(*
Nazwa:			FB_CatchStation
Opis:			Chwytak pod stacjami 
Wersja:			v1.2
Data:			2025-07-08
Autor:			TW,DP
Urzadzenia:		Silownik chwytania, podnośnik JIESANG
Konfiguracja:	
Zmiany:
20250708 - Homing false po wyj. z Manual
20230222 - Zwieksozmny czas bledu 9

Info:
- dodano błędy od nastaw powyżej max i min (error 7 i 8)
- dodawno bHomingNeeded
- wylaczanie wyjść zmiana 2 wylaczanie wyjsc jak zniknie Enable
*)


FUNCTION_BLOCK FB_CatchStation
VAR_INPUT
	bEnable: BOOL;						//Zezwolenie na pracę
	bEStop:BOOL;						//Stop Awaryjny włączony
	bRun:BOOL;							//Rozkaz łapania 
	bHoming:BOOL;						//Zezwolenie na wykonanie bazowania i pozycjonowania podajnika
	bHeightSet:BOOL;					//Ustaw wysokość
	bChangeover:BOOL;					//Ustawianie na zadaną wysokość do wymiany elementów formatowych
	bChangeOver2:BOOL;
	bIgnoreError:BOOL;					//Ignorowania błędów cyklu pracy
	bReset:BOOL;						//Reset błędu, jeśli w stanie "eError"
	nGripperScrewerPosition   	:LREAL; // Aktualna pozycja serwa od podnoszenia
	nSafetyScrewerPosition		:LREAL;	// zadana bezpieczna pozycja 
	bScrewerbError				:BOOL;  // Sygnał błędu od zakręcarki
	nPositionHeightSV:LREAL;			//Wysokość zadana na której ma znajdować się stacja
	bOpenedActuatorSensor:BOOL;			//Czujnik otwarcia siłownika łapania
	bClosedActuatorSensor:BOOL;			//Czujnik otwarcia siłownika łapania
	lrMaxHeight:LREAL;					//Maksymalna wysokość podnośnika chwytaka
	lrMinHeight:LREAL;					//Minimalna wysokość podnośnika chwytaka
	bManualMovement:BOOL;				//Zezwolenie na ruchy ręcznę
	bUnlockColision:BOOL:=FALSE;		//Odblokowywanie możliwośći kolizji
	bAlarmSVCVDiffHeightDisable:BOOL;	//Wyłączenie alarmu od rożnicy wysokości zadanej od aktualnej
	bNoLifter:BOOL;						//Podnośnik
	
	_HEIGHTMOTOR_ :BOOL;	
				
	rHeightMotorPositionOffset :REAL;		//Wysokość bazowani podnośnika
	udiHeightMotorEncoderCV		: UDINT;
	bHeightEncoderSetCDone		: BOOL;	

	_ALARMINFO_ :BOOL;
	iStationIndex:UDINT;					//Numer stacji 
	sStationName:WSTRING;					//Nazwa stacji	

	
END_VAR
VAR_OUTPUT
	eState: E_Station;						//Stan ogólny bloku
	eRunningState: E_CatchStationState;		//Stan wewnętrzny
	bError: BOOL;							//Błąd stacji
	nErrorNr: UDINT;						//Nr błędu podajnika platynek
	sErrorDescription:STRING(200);				//Opis błędu
	sErrorDescription2: STRING(200);				//Opis błędu 2
	sErrorStationName:STRING;				//Nazwa stacji
	udiStationID: UDINT;				// Nr stacji

	bCatchActuator:BOOL;					//Sterownie siłownika łapania opakowania
	bHeightMotorUp:BOOL;					//Sterowanie silnikiem podnośnika  - RUCH W GÓRĘ
	bHeightMotorDown:BOOL;					//Sterowanie silnikiem podnośnika  - RUCH W DÓŁ
	lrHeightMotorCV:LREAL;					//Aktualna pozycja podnośnika
	tCycleTime:TIME;
	bHomingDone:BOOL;						//Wymagane ponowne bazowanie (blad podczas bazowania lub stop awaryjny)
	bCycleDone:BOOL;
	bCycleNotDone:BOOL;
	
				
	udiHeightMotorEncoderSetCV	: UDINT;	
	bHeightEncoderSetC			: BOOL;		

END_VAR
VAR
	tonHeightNoChange: TON; 			//Timer wykrycia braku ruchu siłownika zmiany wysokości stacji
	nLastPositionHeightCV: LREAL;		//Pozycja podnośnika w poprzednim cyklu programu
	tonErrorHeightChange: TON; 			//Timer błędu podnośnika
	// Czas zadziałania siłownika
	tonCatchingTime: TON;
	// Timer blokady otwierania chwytaka
	tonOpeningBlocked: TON;
	rtEncoderHomed:R_TRIG;
	tonCycleTimer:TON;
	rtrigCycleTimerRead:R_TRIG;
	
	tofMotorUpPermition: TOF;
	tofMotorDownPermition: TOF;
	tonLimitPosMinReachedDelay: TON;
	tonLimitPosMaxReachedDelay: TON;
	tonMaxHeight		: TON;
	tonMinHeight		: TON;
	tonSVCVDiffHeight	: TON;
	
	//Podnośnik Jiesang	
	fbHeightMotorEncoder: FB_JiesangActuatorEncoderModul;	// Blok enkodera podnośnika chwytaka stabilizującego pod zakręcarką	
	bHeightMotorEncoderCounterReset:BOOL; 				//Sygnał resetu enkodera
	bHeightMotorEncoderHomed:BOOL;						//Informacja od enkodera że jest zbazowany

	eLastState: E_Station;							//Stan ogólny bloku
	eLastRunningState: E_CatchStationState;			//Stan podbloku
	eLastStateTemp: E_Station;						//Stan ogólny bloku
	eLastRunningStateTemp: E_CatchStationState;		//Stan podbloku
	bStateError: BOOL;

	tonStopping: TON;
	tofHeightMotorDown: TOF;
	iCaseChangeover: INT;
	tonChangeOverLimitPosMinReachedDelay: TON;
	tonChangeoverLimitPosMaxReachedDelay: TON;
	
	//Zmienne od EVENTLOGGER
	bAlarmInit 						: BOOL := TRUE; 
	nAlarmNumerator					: INT;
	arfbAlarm						: ARRAY[0..19] OF  FB_TcAlarm;		//Tablica bloczków błędów
	fbSourceInfo 					: FB_TcSourceInfo;
	iSourceInfo						: I_TcSourceInfo;
	sAlarmTest						: STRING;
	//Koniec zmiennych od EVENTLOGGER
END_VAR

VAR_IN_OUT
	bManualCatchActuator:BOOL;		//Ruch ręczny siłownikiem podajnika platynek
	bManualHeightMotorUp:BOOL;			//Ruch ręczny podnośnika stacji w górę
	bManualHeightMotorDown:BOOL;		//Ruch ręczny podnośnika stacji w dół
END_VAR

HeightMotor();
ErrorHandling();
Control();
Changeover();
Statistics();
aStationID();
(*Zapisywanie ostatniego stanu*)
IF eLastStateTemp<>eState THEN
	eLastState := eLastStateTemp;
END_IF
eLastStateTemp := eState;
IF eLastRunningStateTemp<>eRunningState THEN
	eLastRunningState := eLastRunningStateTemp;
END_IF
eLastRunningStateTemp := eRunningState;
(*Koniec Zapisywanie ostatniego stanu*)


nLastPositionHeightCV:=lrHeightMotorCV;

ACTION aStationID:
udiStationID	:=	iStationIndex;
END_ACTION

ACTION Changeover:
tonChangeOverLimitPosMinReachedDelay(IN:=(lrHeightMotorCV<=lrMinHeight) AND bChangeover,PT:=T#2S);
tonChangeoverLimitPosMaxReachedDelay(IN:=(lrHeightMotorCV>=lrMaxHeight) AND bChangeover,PT:=T#2S);


//Przeniesione do PreparingToDisabled
(*CASE iCaseChangeover OF
	
	0: //Włączenie ustawiania
		IF bChangeover THEN
			iCaseChangeover := iCaseChangeover + 10;
			bHeightMotorDown:=FALSE;
			bHeightMotorUp:=FALSE;
		END_IF
		
	10: //Ustawianie stacji na wysokość 
		IF bHeightMotorEncoderHomed THEN
			bHeightMotorEncoderCounterReset	:=	FALSE;
			bHeightMotorUp					:=	lrHeightMotorCV	<=	200;
			bHeightMotorDown				:=	lrHeightMotorCV	>=	200;
			//Kiedy stacja osiągnie wysokość zadaną
			IF ABS(lrHeightMotorCV-nPositionHeightSV)<2 OR tonChangeoverLimitPosMaxReachedDelay.Q OR tonChangeOverLimitPosMinReachedDelay.Q  THEN
				bHeightMotorDown			:=	FALSE;
				bHeightMotorUp				:=	FALSE;
				iCaseChangeover 			:=	iCaseChangeover + 10;
			END_IF			
		ELSE
			bHeightMotorDown		:=	FALSE;
			bHeightMotorUp			:=	FALSE;
			iCaseChangeover 		:=  0;
		END_IF	
		
	20: //Czekanie na wyłączenie przezbrajania i ustawienie na odpowiednią wysokość z receptury
			IF NOT bChangeover THEN
				iCaseChangeover := iCaseChangeover + 10;
			END_IF
	30: //Ustawianie stacji na wysokość z receptury
		IF bHeightMotorEncoderHomed THEN
			bHeightMotorEncoderCounterReset	:=	FALSE;
			bHeightMotorUp					:=	lrHeightMotorCV	<=	nPositionHeightSV;
			bHeightMotorDown				:=	lrHeightMotorCV	>=	nPositionHeightSV;
			//Kiedy stacja osiągnie wysokość zadaną
			IF ABS(lrHeightMotorCV-nPositionHeightSV)<2 OR tonChangeoverLimitPosMaxReachedDelay.Q OR tonChangeOverLimitPosMinReachedDelay.Q  THEN
				bHeightMotorDown			:=	FALSE;
				bHeightMotorUp				:=	FALSE;
				iCaseChangeover 			:=	iCaseChangeover + 10;
			END_IF			
		ELSE
			bHeightMotorDown		:=	FALSE;
			bHeightMotorUp			:=	FALSE;
			iCaseChangeover 		:=  0;
		END_IF
	40: //Ustawianie stacji na wysokość z receptury	
		iCaseChangeover 		:=  0;

END_CASE
*)
END_ACTION

ACTION Control:

	(** TIMERY**)
	rtEncoderHomed(CLK:=bHeightMotorEncoderHomed,Q=>);
	tonHeightNoChange(IN:=((bHeightMotorUp OR bHeightMotorDown) AND (nLastPositionHeightCV=lrHeightMotorCV)), PT:=T#1S); 
	tonLimitPosMinReachedDelay(IN:=(lrHeightMotorCV<=lrMinHeight) AND eState=E_Station.eHoming,PT:=T#2S);
	tonLimitPosMaxReachedDelay(IN:=(lrHeightMotorCV>=lrMaxHeight) AND eState=E_Station.eHoming,PT:=T#2S);
	tonStopping(IN:=eState=E_Station.eStopping,PT:=T#2S);
	tofMotorUpPermition(IN:=bHeightMotorDown,PT:=T#250MS);
	tofMotorDownPermition(IN:=bHeightMotorUp ,PT:=T#250MS);	
	(*****Wyłączenie enable*****)
	IF NOT bEnable OR bChangeover THEN //Lub przezbrajania
		IF eState <> E_Station.eDisabled AND eState <> E_Station.ePreparingToDisable AND nGripperScrewerPosition>nSafetyScrewerPosition AND NOT bScrewerbError THEN
				eState 				:= E_Station.ePreparingToDisable; 
		END_IF	
	END_IF

	(*****Estop*****)
	IF NOT bEstop  THEN	
		IF eState <> E_Station.eAborted AND eState <> E_Station.eAborting AND eState <> E_Station.eDisabled THEN
				eState 				:= E_Station.eAborting; 
		END_IF
	END_IF

	CASE eState OF
	/////////////////////////////	
		E_Station.eDisabled: 					// Stan nieaktywnosci (Stacja wyłączona) 

			IF bEnable THEN
				eState 				:= E_Station.ePreparingToReady; 
			END_IF 
			
    /////////////////////////////	    
		E_Station.eAborted: 					// Stan bezpiecznego zatrzymania (po Abortingu) 

			IF bEStop THEN
				eState 				:= E_Station.ePreparingToReady;
			END_IF
			
	/////////////////////////////	
		E_Station.eAborting:                 	// Stan bezpiecznego zatrzymywania (po EStopie)

			bHeightMotorUp				:=	FALSE;
			bHeightMotorDown			:=	FALSE;
			eState := E_Station.eAborted;  
			eRunningState:=E_CatchStationState.eDisabled;
			
	/////////////////////////////			
		E_Station.eError:                 	 	// Stan błędu 	

			iCaseChangeover 		:=	0;
			IF bReset THEN
				eState 				:=	E_Station.eResetting;
			END_IF
						
	/////////////////////////////
		E_Station.eResetting:					// Stan resetowania bledu (po Errorze)
	
			bError := FALSE;

			IF NOT bError THEN
				nErrorNr 			:=	0;
   				sErrorDescription 	:=	'';
				eState 				:=	E_Station.ePreparingToReady;
			ELSE
				eState 				:=	E_Station.eError;
			END_IF
        
	/////////////////////////////
		E_Station.eManualMovement:     			// Stan ruchów manualnych  

			ManualMovements();
			//Wyjście z trybu serwisowego
			IF NOT bManualMovement THEN
				IF bHomingDone AND ABS(lrHeightMotorCV - nPositionHeightSV)> 2 THEN
					bHomingDone := FALSE;
				END_IF
				bCatchActuator				:=	FALSE;
				bHeightMotorUp				:=	FALSE;
				bHeightMotorDown			:=	FALSE;
				bManualCatchActuator		:=	bCatchActuator;
				eState:=E_Station.eReady;
			END_IF

	/////////////////////////////
		E_Station.eHoming:						// Stan bazowania 
	IF (nGripperScrewerPosition>nSafetyScrewerPosition AND NOT bScrewerbError) OR bManualMovement THEN  // co to za bzdura
			Homing();
			IF NOT bHoming AND NOT bHeightSet THEN // co to za bzdura
			   eState:=E_Station.ePreparingToReady;
			   	bHeightMotorDown:=FALSE;
				bHeightMotorUp:=FALSE;
			END_IF		
	END_IF		
	/////////////////////////////
		E_Station.eHomingDone:                  // Stan wykonania bazowania 
	
			bHeightMotorDown					:=	FALSE;
			bHeightMotorUp						:=	FALSE;
			bHeightMotorEncoderCounterReset		:=	FALSE;
			bHomingDone							:=	TRUE;
			IF NOT bHoming AND NOT bHeightSet THEN
			   eState:=E_Station.eReady;
			END_IF
			
	/////////////////////////////
		E_Station.ePreparingToReady:            // Stan przygotowywania do gotowosci (zawsze przed Ready)  
	
			bCatchActuator	:=	FALSE;
			eRunningState	:=	E_CatchStationState.eReady;
			eState			:=	E_Station.eReady;	
			
	/////////////////////////////
		E_Station.ePreparingToDisable:          // Stan przygotowywania do nieaktywnosci (po wyłączeniu Enable) 
  
			bCatchActuator:=FALSE;
			IF NOT bChangeOver THEN //Normalne wyłączenie
				bHeightMotorUp:=TRUE;
				bHeightMotorDown:=FALSE;	
				IF tonHeightNoChange.Q THEN
					bHeightMotorUp:=FALSE;
					eState:=E_Station.eDisabled;
					eRunningState:=E_CatchStationState.eDisabled;
				END_IF	
			ELSE //Wyłączenie z przebrajaniem na pozycje 200
				IF bHeightMotorEncoderHomed THEN
					bHeightMotorEncoderCounterReset	:=	FALSE;
					bHeightMotorUp					:=	lrHeightMotorCV	<=	150 AND NOT tofMotorUpPermition.Q;
					bHeightMotorDown				:=	lrHeightMotorCV	>=	150 AND NOT tofMotorDownPermition.Q;
					//Kiedy stacja osiągnie wysokość zadaną
					IF ABS(lrHeightMotorCV-150)<2 OR tonChangeoverLimitPosMaxReachedDelay.Q OR tonChangeOverLimitPosMinReachedDelay.Q  THEN
						bHeightMotorDown			:=	FALSE;
						bHeightMotorUp				:=	FALSE;
						eState						:=	E_Station.eDisabled;
						eRunningState				:=	E_CatchStationState.eDisabled;
					END_IF			
				ELSE
					bHeightMotorDown				:=	FALSE;
					bHeightMotorUp					:=	FALSE;
					eState								:=E_Station.eDisabled;
					eRunningState					:=	E_CatchStationState.eDisabled;
				END_IF	
			END_IF
				
	/////////////////////////////
		E_Station.eReady:						// Stan gotowosci 

			IF bRun AND NOT bCycleDone AND NOT bCycleNotDone THEN
				eState 				:= E_Station.eStarting; 
			END_IF
			IF bHoming OR bHeightSet OR bChangeover THEN
				eState 				:= E_Station.eHoming; 
			END_IF
			IF bManualMovement THEN
				//Jeśli przejście w tryb ruchów manualnych przepisz wszystkie stany siłowników sterowanych przez moduł
				//aby zapobiec ewentualnym kolizjom po wejściu w tryb serwisowy
				bManualCatchActuator		:= bCatchActuator;
				bManualHeightMotorUp		:= bHeightMotorUp;
				bManualHeightMotorDown		:= bHeightMotorDown;
				
				eState 						:= E_Station.eManualMovement; 
				eRunningState 				:= E_CatchStationState.eReady;
 
			END_IF
			IF NOT bRun THEN
				bCycleDone 			:= FALSE;
				bCycleNotDone 		:= FALSE;			
			END_IF
			
	/////////////////////////////
		E_Station.eStopping:					// Stan zatrzymywania 
					
			Running();
			IF bOpenedActuatorSensor OR tonStopping.Q THEN //NEW
				eState						:=	E_Station.eReady;
				eRunningState 				:=	E_CatchStationState.eReady;
			END_IF
			
	/////////////////////////////
		E_Station.eStarting:                  	// Stan uruchamiania (po Ready)
				
			eState					 := E_Station.eRunning; 

	/////////////////////////////
		E_Station.eRunning:               		// Stan wykonywania cyklu (po Startingu), w tym stanie osobny

			Running();
			IF NOT bRun THEN 					(*Przerywanie cyklu*)
				eState				:= E_Station.eStopping;
				bCycleNotDone		:= TRUE;
			END_IF
			(*IF bCycleDone OR bCycleNotDone THEN (*Cykl zakończony*)
				eState 				 := E_Station.eReady;
			END_IF*)						
		ELSE
		
		
	/////////////////////////////		
	END_CASE
END_ACTION

ACTION ErrorHandling:
// Alarm_0440	440	Error	Blokada otwarcia chwytaka - sprawdź czujnik
// Alarm_0441	441	Error	Blokada podnośnika lub brak zasilania - sprawdź czujnik lub odblokuj mechanicznie
// Alarm_0442	442	Error	Wartość zadana wysokości jest większa od maksymalnej - zmień ustawienia w recepturze {0}
// Alarm_0443	443	Error	Wartość zadana wysokości jest mniejsza od minimalnej - zmień ustawienia w recepturze {0}
// Alarm_0444	444	Error	Wartość aktualna jest zbyt różna od zadanej - zmień ustawienia w recepturze lub ustaw stację

IF bAlarmInit THEN
    bAlarmInit := FALSE; 
	fbSourceInfo.Clear();
	fbSourceInfo.sName:=wsLiteral_TO_UTF8(sStationName);//'Machine';
	fbSourceInfo.nId:=iStationIndex;//2700;
	// Alarm_0440	440	Error	Blokada otwarcia chwytaka - sprawdź czujnik
    arfbAlarm[0].CreateEx(stEventEntry := TC_EVENTS.AlarmClass.Alarm_0440, bWithConfirmation:= FALSE,  ipSourceInfo:= fbSourceInfo); 
	// Alarm_0441	441	Error	Blokada podnośnika lub brak zasilania - sprawdź czujnik lub odblokuj mechanicznie
	arfbAlarm[1].CreateEx(stEventEntry := TC_EVENTS.AlarmClass.Alarm_0441, bWithConfirmation:= FALSE,  ipSourceInfo:= fbSourceInfo);
	// Alarm_0442	442	Error	Wartość zadana wysokości jest większa od maksymalnej - zmień ustawienia w recepturze {0}
	arfbAlarm[2].CreateEx(stEventEntry := TC_EVENTS.AlarmClass.Alarm_0442, bWithConfirmation:= FALSE,  ipSourceInfo:= fbSourceInfo);
	// Alarm_0443	443	Error	Wartość zadana wysokości jest mniejsza od minimalnej - zmień ustawienia w recepturze {0}
	arfbAlarm[3].CreateEx(stEventEntry := TC_EVENTS.AlarmClass.Alarm_0443, bWithConfirmation:= FALSE,  ipSourceInfo:= fbSourceInfo);
	// Alarm_0444	444	Error	Wartość aktualna jest zbyt różna od zadanej - zmień ustawienia w recepturze lub ustaw stację
	arfbAlarm[4].CreateEx(stEventEntry := TC_EVENTS.AlarmClass.Alarm_0444, bWithConfirmation:= FALSE,  ipSourceInfo:= fbSourceInfo);
END_IF

//OBSŁUGA BŁĘDÓW PODAJNIKA PLATYNEK

//************LISTA BŁĘDÓW***************
bStateError:= (eState=E_Station.eError) OR (eState=E_Station.eResetting) OR bIgnoreError;




IF bEnable THEN
	// Alarm_0440	440	Error	Blokada otwarcia chwytaka - sprawdź czujnik
	//Error 1 - Blokada otwarcia chwytaka
	tonOpeningBlocked(IN:=NOT bCatchActuator AND NOT bOpenedActuatorSensor, PT:=T#3S);
	
	IF tonOpeningBlocked.Q THEN
		IF NOT arfbAlarm[0].bActive THEN
			arfbAlarm[0].Raise(nTimeStamp:=0);
		END_IF
	ELSE	
		IF  arfbAlarm[0].bActive AND bReset THEN
			arfbAlarm[0].Clear(nTimeStamp:=0, bResetConfirmation:= FALSE);
		END_IF
// 		sErrorDescription:='Blokada otwarcia chwytaka - sprawdź czujnik';
// 		bHeightMotorUp:=FALSE;
// 		bError := TRUE;
// 		nErrorNr:=281;	
// 		//nErrorNr := nErrorNr+iStationIndex;
	END_IF
	// Alarm_0441	441	Error	Blokada podnośnika lub brak zasilania - sprawdź czujnik lub odblokuj mechanicznie
	//Error 2 - podnośnik nie porusza się pomimo wysterowania 
	tonErrorHeightChange(IN:=(bHeightMotorUp OR bHeightMotorDown) AND nLastPositionHeightCV=lrHeightMotorCV AND NOT bNoLifter, PT:=T#3S);
	
	IF tonErrorHeightChange.Q THEN
		IF NOT arfbAlarm[1].bActive THEN
			bHeightMotorUp:=FALSE;
			bHeightMotorDown:=FALSE;
			arfbAlarm[1].Raise(nTimeStamp:=0);
		END_IF
	ELSE	
		IF  arfbAlarm[1].bActive AND bReset THEN
			arfbAlarm[1].Clear(nTimeStamp:=0, bResetConfirmation:= FALSE);
		END_IF
// 		bHeightMotorUp:=FALSE;
// 		bHeightMotorDown:=FALSE;
// 		bError := TRUE;
// 		nErrorNr:=282;
// 		//nErrorNr := nErrorNr+iStationIndex;
// 		sErrorDescription:='Blokada podnośnika lub brak zasilania - sprawdź czujnik lub odblokuj mechanicznie';	
	END_IF
	
	// Alarm_0442	442	Error	Wartość zadana wysokości jest większa od maksymalnej - zmień ustawienia w recepturze {0}
	//Error 3 - Bład nastaw max
	tonMaxHeight(IN:=nPositionHeightSV>lrMaxHeight+1 AND bHomingDone AND lrMaxHeight>0 AND eState=E_Station.eReady,PT:=T#30S);
	IF tonMaxHeight.Q THEN
		arfbAlarm[2].ipArguments.Clear() .AddLReal(lrMaxHeight);
		IF NOT arfbAlarm[2].bActive THEN
			bHeightMotorUp:=FALSE;
			bHeightMotorDown:=FALSE;
			arfbAlarm[2].Raise(nTimeStamp:=0);
		END_IF
	ELSE	
		IF  arfbAlarm[2].bActive AND bReset THEN
			arfbAlarm[2].Clear(nTimeStamp:=0, bResetConfirmation:= FALSE);
		END_IF	
// 		bHeightMotorUp:=FALSE;
// 		bHeightMotorDown:=FALSE;
// 		bError := TRUE;
// 		nErrorNr:=283;
// 		//nErrorNr := nErrorNr+iStationIndex;
// 		sErrorDescription:='Wartość zadana wysokości jest większa od maksymalnej - zmień ustawienia w recepturze';
// 		sErrorDescription2:=REAL_TO_STRING(LREAL_TO_INT(lrMaxHeight));
	END_IF
	// Alarm_0443	443	Error	Wartość zadana wysokości jest mniejsza od minimalnej - zmień ustawienia w recepturze {0}
	//Error 4 - Bład nastaw min
	tonMinHeight(IN:=nPositionHeightSV<lrMinHeight-1 AND bHomingDone AND lrMinHeight>0 AND eState=E_Station.eReady,PT:=T#30S);
	IF tonMinHeight.Q THEN
		arfbAlarm[3].ipArguments.Clear() .AddLReal(lrMinHeight);
		IF NOT arfbAlarm[3].bActive THEN
			bHeightMotorUp:=FALSE;
			bHeightMotorDown:=FALSE;
			arfbAlarm[3].Raise(nTimeStamp:=0);
		END_IF
	ELSE	
		IF  arfbAlarm[3].bActive AND bReset THEN
			arfbAlarm[3].Clear(nTimeStamp:=0, bResetConfirmation:= FALSE);
		END_IF
// 		bHeightMotorUp:=FALSE;
// 		bHeightMotorDown:=FALSE;
// 		bError := TRUE;
// 		nErrorNr:=284;
// 		//nErrorNr := nErrorNr+iStationIndex;
// 		sErrorDescription:='Wartość zadana wysokości jest mniejsza od minimalnej - zmień ustawienia w recepturze ';
// 		sErrorDescription2:=REAL_TO_STRING(LREAL_TO_INT(lrMinHeight));
	END_IF
	// Alarm_0444	444	Error	Wartość aktualna jest zbyt różna od zadanej - zmień ustawienia w recepturze lub ustaw stację
	//Error 5 - Bład zbyt dużej różnicy nastaw
	//tonSVCVDiffHeight(IN:=ABS(nPositionHeightSV-lrHeightMotorCV)>10 AND bHomingDone AND NOT bAlarmSVCVDiffHeightDisable AND eState=E_Station.eReady AND NOT bChangeOver2,PT:=T#5M);
	IF tonSVCVDiffHeight.Q THEN
		arfbAlarm[4].ipArguments.Clear() .AddLReal(nPositionHeightSV);
		IF NOT arfbAlarm[4].bActive THEN
			bHeightMotorUp:=FALSE;
			bHeightMotorDown:=FALSE;
			arfbAlarm[4].Raise(nTimeStamp:=0);
		END_IF
	ELSE	
		IF  arfbAlarm[4].bActive AND bReset THEN
			arfbAlarm[4].Clear(nTimeStamp:=0, bResetConfirmation:= FALSE);
		END_IF
// 		bHeightMotorUp:=FALSE;
// 		bHeightMotorDown:=FALSE;
// 		bError := TRUE;
// 		nErrorNr:=285;
// 		//nErrorNr := nErrorNr+iStationIndex;
// 		sErrorDescription:='Wartość aktualna jest zbyt różna od zadanej - zmień ustawienia w recepturze lub ustaw stację';
// 		sErrorDescription2:=REAL_TO_STRING(LREAL_TO_INT(nPositionHeightSV));
		
	END_IF	
		
	
	
ELSE
	bError := FALSE;
END_IF

	
//******************PRZEJŚCIE DO eERROR*****************************

IF bError AND NOT bStateError THEN
	IF eLastState = eRunning THEN
		bCycleNotDone := TRUE;
	END_IF
	eState := E_Station.eError;
END_IF

//****************WYŚWIETLANIE STATUSU BLEDU***********************

(*Wyświetlanie błedu na wyjściu*)
bError							:= FALSE;
FOR nAlarmNumerator := 0 TO 19 DO
	bError						:= bError OR arfbAlarm[nAlarmNumerator].bActive;
END_FOR

(*Przepisywanie nazwy stacji*)
sErrorStationName := WSTRING_TO_STRING(sStationName);


//Jezeli nie zbazowane to potrzebne bazowanie
IF NOT bHeightMotorEncoderHomed AND NOT bNoLifter  THEN
	bHomingDone:=FALSE;
END_IF
END_ACTION

ACTION HeightMotor:
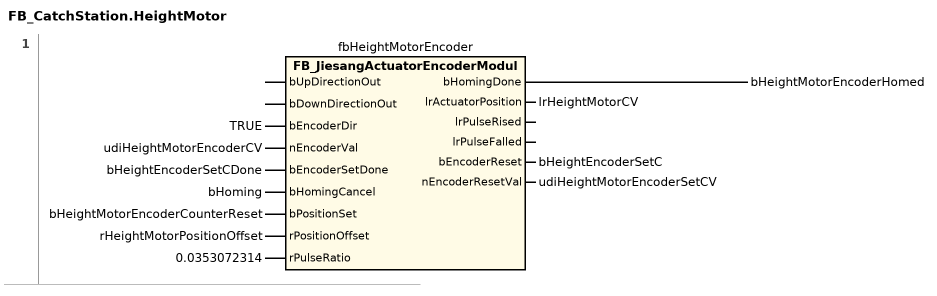
// NETWORK 1
fbHeightMotorEncoder(
    bEncoderDir := TRUE,
    nEncoderVal := udiHeightMotorEncoderCV,
    bEncoderSetDone := bHeightEncoderSetCDone,
    bHomingCancel := bHoming,
    bPositionSet := bHeightMotorEncoderCounterReset,
    rPositionOffset := rHeightMotorPositionOffset,
    rPulseRatio := 0.0353072314,
    lrActuatorPosition => lrHeightMotorCV,
    bEncoderReset => bHeightEncoderSetC,
    nEncoderResetVal => udiHeightMotorEncoderSetCV); // FB_JiesangActuatorEncoderModul
bHeightMotorEncoderHomed := fbHeightMotorEncoder.bHomingDone;
END_ACTION

ACTION Homing:
//BAZOWANIE
bCatchActuator:=FALSE;
	
//Uwaga nie zmieniać czasu bo jednocześnie dwie stację jadą do góry
tofHeightMotorDown(IN:=bHeightMotorDown, PT:=T#1S); //Zabezpieczenie przed zbyt szybkim przełączeniem pomiędzy Down a Up, bezpiecznieki sie palą, 


//Podnoszenie stacji do maksymalnej pozycji
IF NOT bHeightMotorEncoderHomed OR rtEncoderHomed.Q THEN
	bHeightMotorUp:=(*TRUE*) NOT tofHeightMotorDown.Q;;
	bHeightMotorDown:=FALSE;
	IF tonHeightNoChange.Q THEN
		bHeightMotorEncoderCounterReset:=TRUE;
		bHeightMotorUp:=FALSE;
	END_IF
	//Jesli enkoder zbazowany zakończ bazowanie	
	IF rtEncoderHomed.Q THEN
		bHeightMotorUp:=FALSE;
		bHeightMotorDown:=FALSE;
		eState:=E_Station.eHomingDone;
	END_IF		
		
//Po podniesieniu stacji opuszczanie do ustalonej wysokości
ELSIF bHeightMotorEncoderHomed THEN
	bHeightMotorEncoderCounterReset:=FALSE;
	bHeightMotorUp:=lrHeightMotorCV<=nPositionHeightSV;
	bHeightMotorDown:=lrHeightMotorCV>=nPositionHeightSV (*AND lrHeightMotorCV>=lrMinHeight*);
	//Kiedy stacja osiągnie wysokość zadaną
	IF ABS(lrHeightMotorCV-nPositionHeightSV)<1 OR tonLimitPosMaxReachedDelay.Q OR tonLimitPosMinReachedDelay.Q (*OR lrHeightMotorCV>=lrMinHeight*) THEN
		bHeightMotorDown:=FALSE;
		bHeightMotorUp:=FALSE;
		eState:=E_Station.eHomingDone;
	END_IF			
END_IF

	
//Opcja braku podnośnika	
IF bNoLifter THEN
	eState:=E_Station.eHomingDone;
END_IF
END_ACTION

ACTION ManualMovements:

//W trybie ruchów manualnych wykonuj ruchy za pomocą rozkazów manualnych
IF NOT bRun THEN
	bCatchActuator:=bManualCatchActuator;
	bHeightMotorUp:=bManualHeightMotorUp;
	bHeightMotorDown:=bManualHeightMotorDown;
ELSE	//Kasuje zeby po cyklu nic sie nie poruszało
	bManualCatchActuator := FALSE;
	bManualHeightMotorUp  := FALSE;
	bManualHeightMotorDown  := FALSE;
END_IF


IF bHoming OR bHeightSet THEN
	eState:=E_Station.eHoming;
END_IF
	
Running();
	
//Zabezpieczenie przed kolizją stacji poprzez ruch podnośnika	
IF bHeightMotorDown AND lrHeightMotorCV<=lrMinHeight AND NOT bHoming AND NOT bHeightSet THEN
	bHeightMotorDown:=FALSE;
END_IF	

IF bHeightMotorUp AND lrHeightMotorCV>=lrMaxHeight AND NOT bHoming AND NOT bHeightSet THEN
	bHeightMotorUp:=FALSE;
END_IF		 

IF NOT bRun THEN
	bCycleDone 					:= FALSE;
	bCycleNotDone 				:= FALSE;	
END_IF
END_ACTION

ACTION Running:

//Timery
tonCatchingTime(IN:=(eRunningState=E_CatchStationState.eCatching), PT:=T#500MS);


CASE eRunningState OF
	
	//NIEGOTOWY
	E_CatchStationState.eDisabled:
		eRunningState:=E_CatchStationState.eReady;

	//Chwytak gotowy do pracy
	E_CatchStationState.eReady: 
		//Jeśli komenda chwytania przejdz do stanu chwytanie
		IF NOT bCycleDone AND NOT bCycleNotDone THEN
			IF bRun THEN
			eRunningState:=E_CatchStationState.eCatching;
			END_IF
		END_IF
		
	//Chwytanie 
	E_CatchStationState.eCatching:
		bCatchActuator:=TRUE;
		

		IF tonCatchingTime.Q THEN
			IF bClosedActuatorSensor THEN
				eRunningState	:= E_CatchStationState.eCatched;
			ELSE
				eRunningState	:= E_CatchStationState.eNotCatched;
			END_IF
		END_IF

	//Uchwycone 
	E_CatchStationState.eCatched:
		bCatchActuator:=bRun;
		bCycleDone := TRUE;
		//Kiedy zniknie rozkaz chwytania i 
	
	E_CatchStationState.eNotCatched:
	
		bCatchActuator:=bRun;                                   
		bCycleDone := TRUE;
	
END_CASE
END_ACTION

ACTION Statistics:



rtrigCycleTimerRead(CLK:=eRunningState=E_CatchStationState.eCatched);
IF rtrigCycleTimerRead.Q THEN
	tCycleTime:=tonCycleTimer.ET;
END_IF
tonCycleTimer(IN:=eState>E_Station.eReady,PT:=T#1D);
END_ACTION

END_FUNCTION_BLOCK

(* stored: Version 1.1.0.1, ProductVersion 3.1.4026.13, FileIdentifier 9de2814f4a6887c84a943f926182f0d1dfaf98cc, FileSignature 71c145b576d1383769d172a182114cc93fda9e059769a4f1549fcbaee4e510ca71e4c732371450b83b2c373a464b095f86e5eb7b043b2bd4f9dca8e7172eb4db855658ffd6a8ccfe13f622959784d7e1a7c709996711eec6a9c4c9c6964df99311a60f68e058162329a2e2ff8c49ce848424f5474edf49ad08ba59d1f9b13075504695641cdd7cd733106635462a2410c16a00aaf1f019ebc564e4253a199f4730a6fc56e25294102f1533f483c36037433ea508e2b6f5f5e385b643a5912c8a496999bcbe3695ccd668ed49567e4da13a8dbece4fe5af04702670ac725b2b0fcbb3dceffa0d86f99856753ae9606fae73b8d5b7df5a8287164ae54c0313ad0b
   POU FB_CatchStation: Id {0e7ba2fc-097d-4c24-856f-cc572bc2d435}, SpecialFunc None
   Action aStationID: Id {f538eae6-c229-4871-8d1e-9fe88a2bdf79}
   Action Changeover: Id {50310c47-4347-4143-b980-61468f307ab3}
   Action Control: Id {9cadcbbd-7e42-4184-8dae-e25cfe7f3a5f}
   Action ErrorHandling: Id {3fd0bd17-f0ee-4720-92fa-0ccc788777cc}
   Action HeightMotor: Id {401744c5-adab-4a66-a5fe-36545824055a}
   Action Homing: Id {61327328-d689-47a5-ba8f-bc31300485fa}
   Action ManualMovements: Id {771e4f2d-f10e-4bff-aced-cc88991b62db}
   Action Running: Id {b9043bdf-5c3e-4029-a2e6-1c7c7827b727}
   Action Statistics: Id {5d07f1af-c568-4c5c-81ac-6607d9c06cf7} *)
